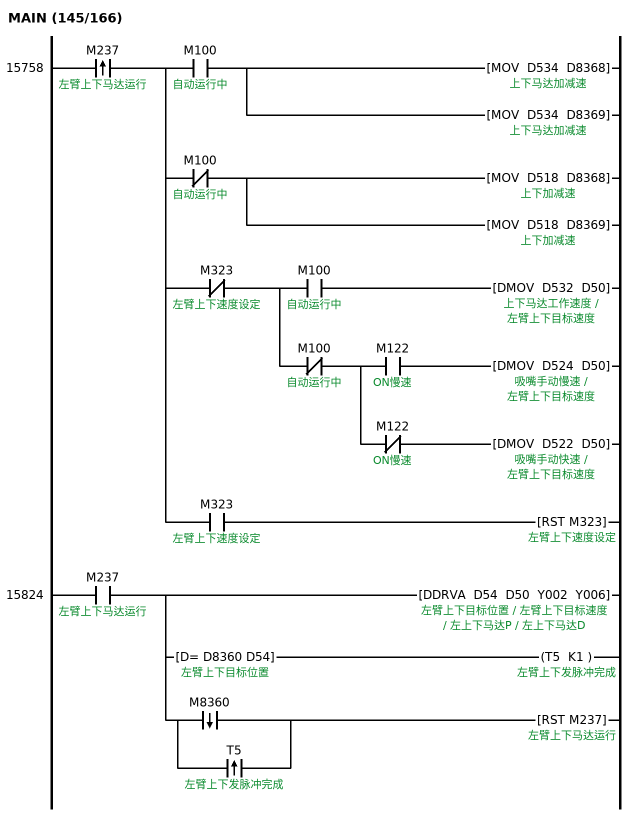
[picture p144: ladder of MAIN, rungs at steps 15758 to 15824]
15758 LDP     M237  ; 左臂上下马达运行
      MPS
      AND     M100  ; 自动运行中
      MOV     D534 D8368
      MOV     D534 D8369
      MRD
      ANI     M100  ; 自动运行中
      MOV     D518 D8368
      MOV     D518 D8369
      MRD
      ANI     M323  ; 左臂上下速度设定
      MPS
      AND     M100  ; 自动运行中
      DMOV    D532 D50
      MPP
      ANI     M100  ; 自动运行中
      MPS
      AND     M122  ; ON慢速
      DMOV    D524 D50
      MPP
      ANI     M122  ; ON慢速
      DMOV    D522 D50
      MPP
      AND     M323  ; 左臂上下速度设定
      RST     M323  ; 左臂上下速度设定
15824 LD      M237  ; 左臂上下马达运行
      DDRVA   D54 D50 Y002 Y006  ; 左上下马达P / 左上下马达D
      MPS
      ANDD=   D8360 D54  ; 左臂上下目标位置
      OUT     T5 K1  ; 左臂上下发脉冲完成
      MPP
      LDF     M8360
      ORP     T5  ; 左臂上下发脉冲完成
      ANB
      RST     M237  ; 左臂上下马达运行
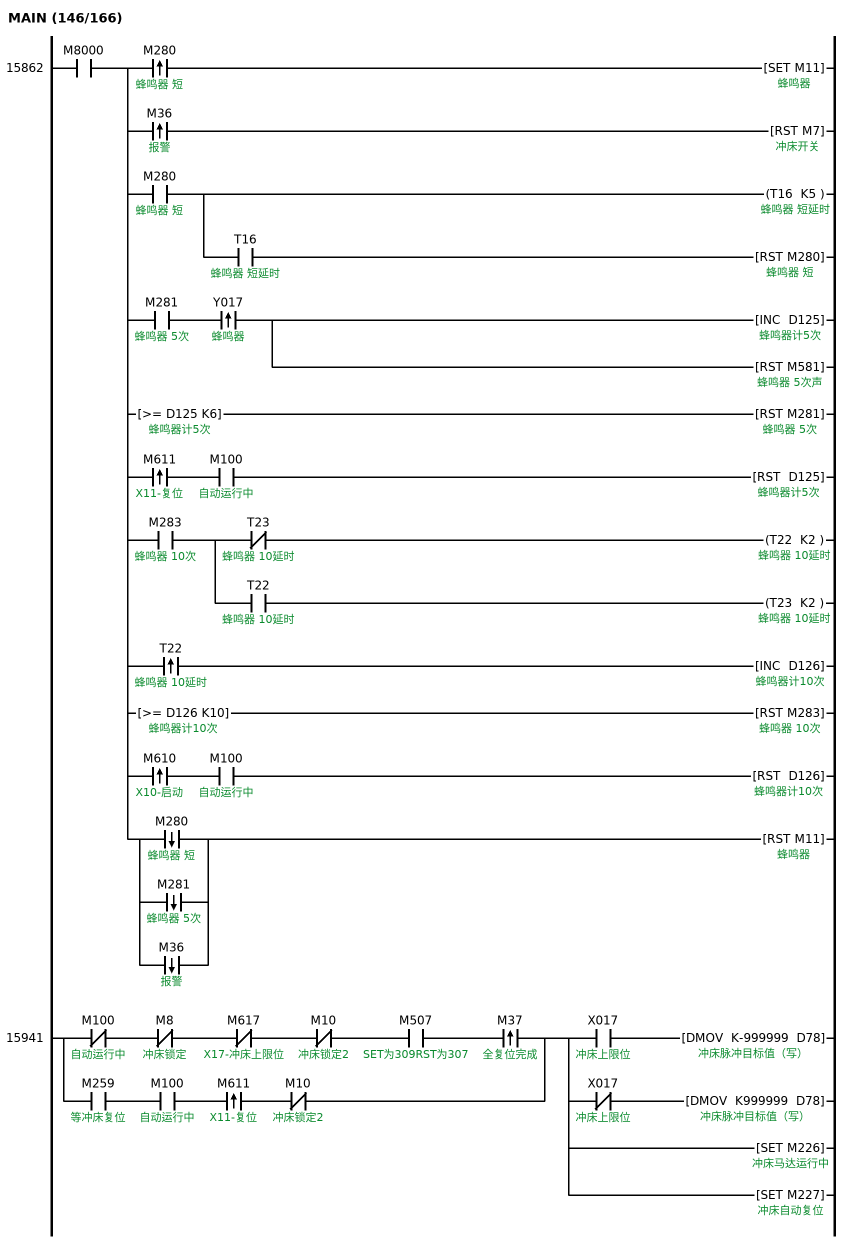
15862 LD      M8000
      MPS
      ANDP    M280  ; 蜂鸣器 短
      SET     M11  ; 蜂鸣器
      MRD
      ANDP    M36  ; 报警
      RST     M7  ; 冲床开关
      MRD
      AND     M280  ; 蜂鸣器 短
      OUT     T16 K5  ; 蜂鸣器 短延时
      AND     T16  ; 蜂鸣器 短延时
      RST     M280  ; 蜂鸣器 短
      MRD
      AND     M281  ; 蜂鸣器 5次
      ANDP    Y017  ; 蜂鸣器
      INC     D125
      RST     M581  ; 蜂鸣器 5次声
      MRD
      AND>=   D125 K6  ; 蜂鸣器计5次
      RST     M281  ; 蜂鸣器 5次
      MRD
      ANDP    M611  ; X11-复位
      AND     M100  ; 自动运行中
      RST     D125  ; 蜂鸣器计5次
      MRD
      AND     M283  ; 蜂鸣器 10次
      MPS
      ANI     T23  ; 蜂鸣器 10延时
      OUT     T22 K2  ; 蜂鸣器 10延时
      MPP
      AND     T22  ; 蜂鸣器 10延时
      OUT     T23 K2  ; 蜂鸣器 10延时
      MRD
      ANDP    T22  ; 蜂鸣器 10延时
      INC     D126  ; 蜂鸣器计10次
      MRD
      AND>=   D126 K10  ; 蜂鸣器计10次
      RST     M283  ; 蜂鸣器 10次
      MRD
      ANDP    M610  ; X10-启动
      AND     M100  ; 自动运行中
      RST     D126  ; 蜂鸣器计10次
      MPP
      LDF     M280  ; 蜂鸣器 短
      ORF     M281  ; 蜂鸣器 5次
      ORF     M36  ; 报警
      ANB
      RST     M11  ; 蜂鸣器
15941 LDI     M100  ; 自动运行中
      ANI     M8  ; 冲床锁定
      ANI     M617  ; X17-冲床上限位
      ANI     M10  ; 冲床锁定2
      AND     M507  ; SET为309RST为307
      ANDP    M37  ; 全复位完成
      LD      M259  ; 等冲床复位
      AND     M100  ; 自动运行中
      ANDP    M611  ; X11-复位
      ANI     M10  ; 冲床锁定2
      ORB
      MPS
      AND     X017  ; 冲床上限位
      DMOV    K-999999 D78  ; 冲床脉冲目标值（写）
      MRD
      ANI     X017  ; 冲床上限位
      DMOV    K999999 D78
      MPP
      SET     M226  ; 冲床马达运行中
      SET     M227  ; 冲床自动复位
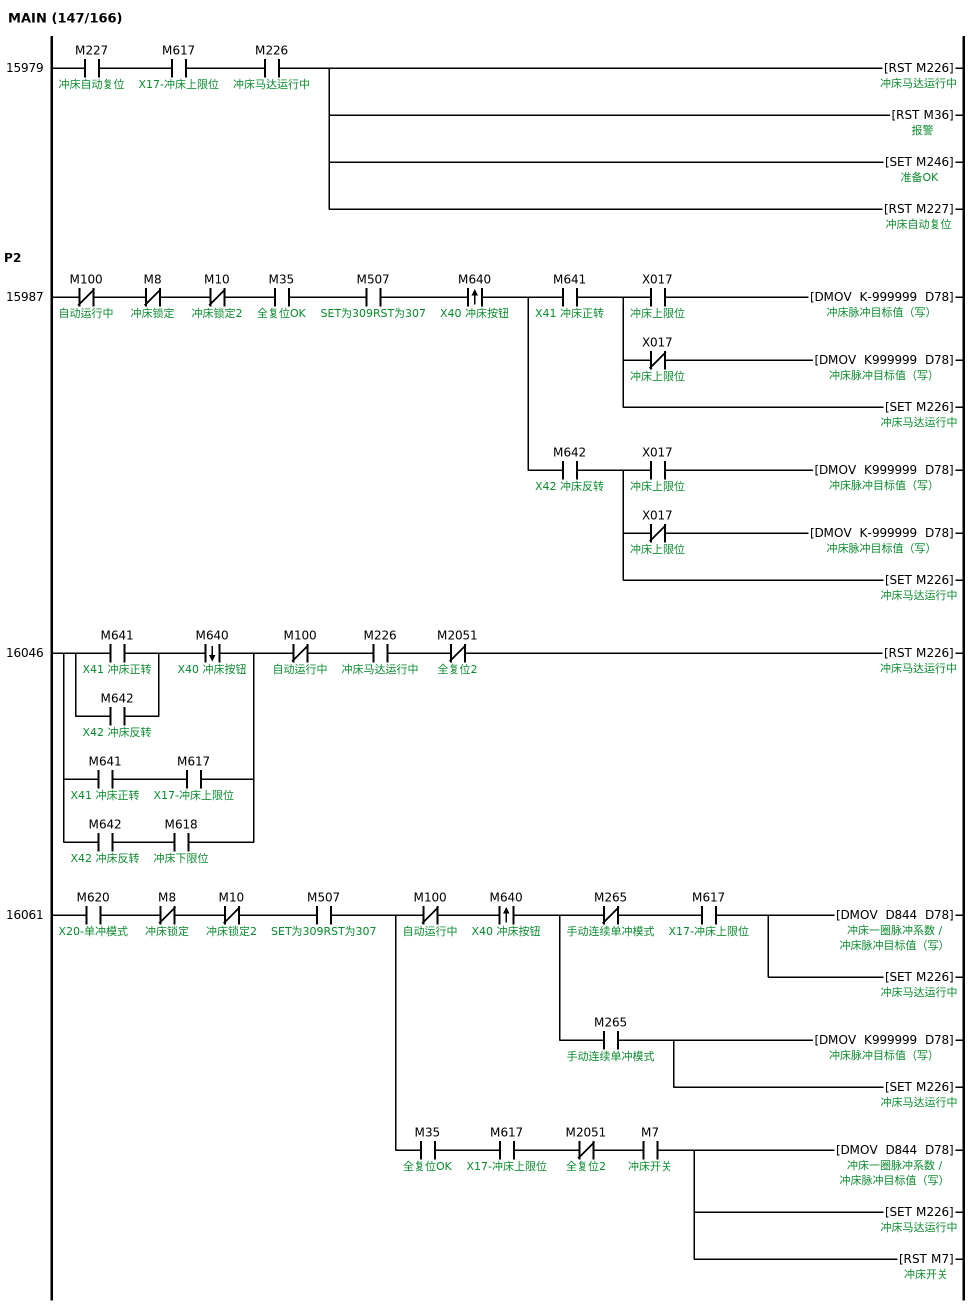
15979 LD      M227  ; 冲床自动复位
      AND     M617  ; X17-冲床上限位
      AND     M226  ; 冲床马达运行中
      RST     M226  ; 冲床马达运行中
      RST     M36  ; 报警
      SET     M246  ; 准备OK
      RST     M227  ; 冲床自动复位
      P2
15987 LDI     M100  ; 自动运行中
      ANI     M8  ; 冲床锁定
      ANI     M10  ; 冲床锁定2
      AND     M35  ; 全复位OK
      AND     M507  ; SET为309RST为307
      ANDP    M640  ; X40 冲床按钮
      MPS
      AND     M641  ; X41 冲床正转
      MPS
      AND     X017  ; 冲床上限位
      DMOV    K-999999 D78
      MRD
      ANI     X017  ; 冲床上限位
      DMOV    K999999 D78
      MPP
      SET     M226  ; 冲床马达运行中
      MPP
      AND     M642  ; X42 冲床反转
      MPS
      AND     X017  ; 冲床上限位
      DMOV    K999999 D78
      MRD
      ANI     X017  ; 冲床上限位
      DMOV    K-999999 D78
      MPP
      SET     M226  ; 冲床马达运行中
16046 LD      M641  ; X41 冲床正转
      OR      M642  ; X42 冲床反转
      ANDF    M640  ; X40 冲床按钮
      LD      M641  ; X41 冲床正转
      AND     M617  ; X17-冲床上限位
      ORB
      LD      M642  ; X42 冲床反转
      AND     M618  ; 冲床下限位
      ORB
      ANI     M100  ; 自动运行中
      AND     M226  ; 冲床马达运行中
      ANI     M2051  ; 全复位2
      RST     M226  ; 冲床马达运行中
16061 LD      M620  ; X20-单冲模式
      ANI     M8  ; 冲床锁定
      ANI     M10  ; 冲床锁定2
      AND     M507  ; SET为309RST为307
      MPS
      ANI     M100  ; 自动运行中
      ANDP    M640  ; X40 冲床按钮
      MPS
      ANI     M265  ; 手动连续单冲模式
      AND     M617  ; X17-冲床上限位
      DMOV    D844 D78
      SET     M226  ; 冲床马达运行中
      MPP
      AND     M265  ; 手动连续单冲模式
      DMOV    K999999 D78
      SET     M226  ; 冲床马达运行中
      MPP
      AND     M35  ; 全复位OK
      AND     M617  ; X17-冲床上限位
      ANI     M2051  ; 全复位2
      AND     M7  ; 冲床开关
      DMOV    D844 D78
      SET     M226  ; 冲床马达运行中
      RST     M7  ; 冲床开关
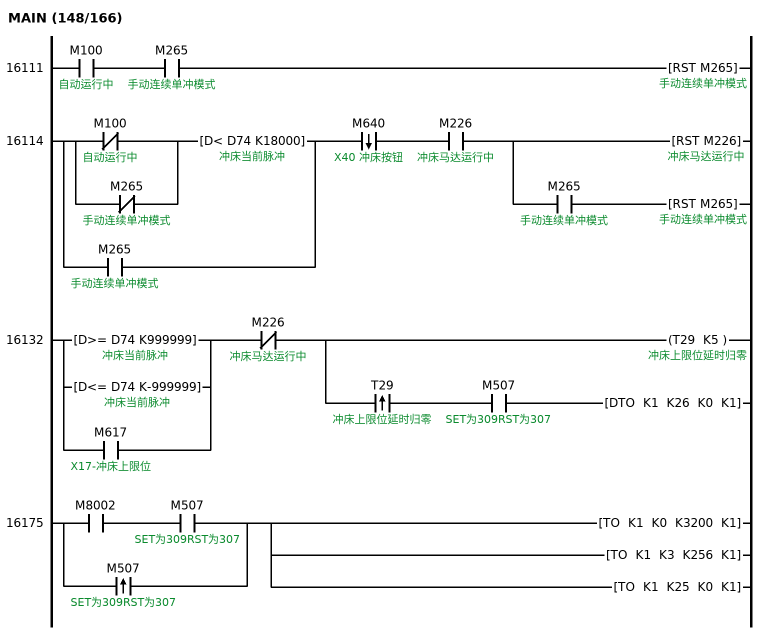
16111 LD      M100  ; 自动运行中
      AND     M265  ; 手动连续单冲模式
      RST     M265  ; 手动连续单冲模式
16114 LDI     M100  ; 自动运行中
      ORI     M265  ; 手动连续单冲模式
      ANDD<   D74 K18000  ; 冲床当前脉冲
      OR      M265  ; 手动连续单冲模式
      ANDF    M640  ; X40 冲床按钮
      AND     M226  ; 冲床马达运行中
      RST     M226  ; 冲床马达运行中
      AND     M265  ; 手动连续单冲模式
      RST     M265  ; 手动连续单冲模式
16132 LDD>=   D74 K999999  ; 冲床当前脉冲
      ORD<=   D74 K-999999  ; 冲床当前脉冲
      OR      M617  ; X17-冲床上限位
      ANI     M226  ; 冲床马达运行中
      OUT     T29 K5  ; 冲床上限位延时归零
      ANDP    T29  ; 冲床上限位延时归零
      AND     M507  ; SET为309RST为307
      DTO     K1 K26 K0 K1
16175 LD      M8002
      AND     M507  ; SET为309RST为307
      ORP     M507  ; SET为309RST为307
      TO      K1 K0 K3200 K1
      TO      K1 K3 K256 K1
      TO      K1 K25 K0 K1
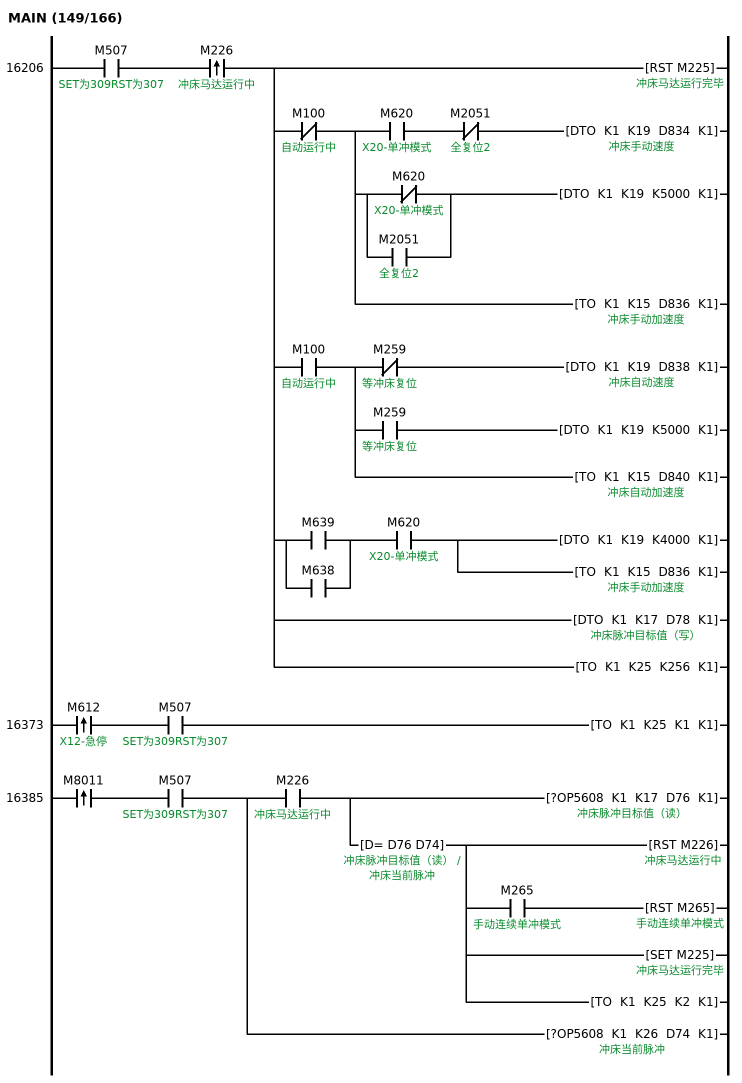
16206 LD      M507  ; SET为309RST为307
      ANDP    M226  ; 冲床马达运行中
      RST     M225  ; 冲床马达运行完毕
      MPS
      ANI     M100  ; 自动运行中
      MPS
      AND     M620  ; X20-单冲模式
      ANI     M2051  ; 全复位2
      DTO     K1 K19 D834 K1
      MRD
      LDI     M620  ; X20-单冲模式
      OR      M2051  ; 全复位2
      ANB
      DTO     K1 K19 K5000 K1
      MPP
      TO      K1 K15 D836 K1
      MRD
      AND     M100  ; 自动运行中
      MPS
      ANI     M259  ; 等冲床复位
      DTO     K1 K19 D838 K1
      MRD
      AND     M259  ; 等冲床复位
      DTO     K1 K19 K5000 K1
      MPP
      TO      K1 K15 D840 K1
      MRD
      LD      M639
      OR      M638
      ANB
      AND     M620  ; X20-单冲模式
      DTO     K1 K19 K4000 K1
      TO      K1 K15 D836 K1
      MPP
      DTO     K1 K17 D78 K1
      TO      K1 K25 K256 K1
16373 LDP     M612  ; X12-急停
      AND     M507  ; SET为309RST为307
      TO      K1 K25 K1 K1
16385 LDP     M8011
      AND     M507  ; SET为309RST为307
      MPS
      AND     M226  ; 冲床马达运行中
      ?OP5608 K1 K17 D76 K1  ; 冲床脉冲目标值（读）
      ANDD=   D76 D74  ; 冲床脉冲目标值（读） / 冲床当前脉冲
      RST     M226  ; 冲床马达运行中
      MPS
      AND     M265  ; 手动连续单冲模式
      RST     M265  ; 手动连续单冲模式
      MPP
      SET     M225  ; 冲床马达运行完毕
      TO      K1 K25 K2 K1
      MPP
      ?OP5608 K1 K26 D74 K1
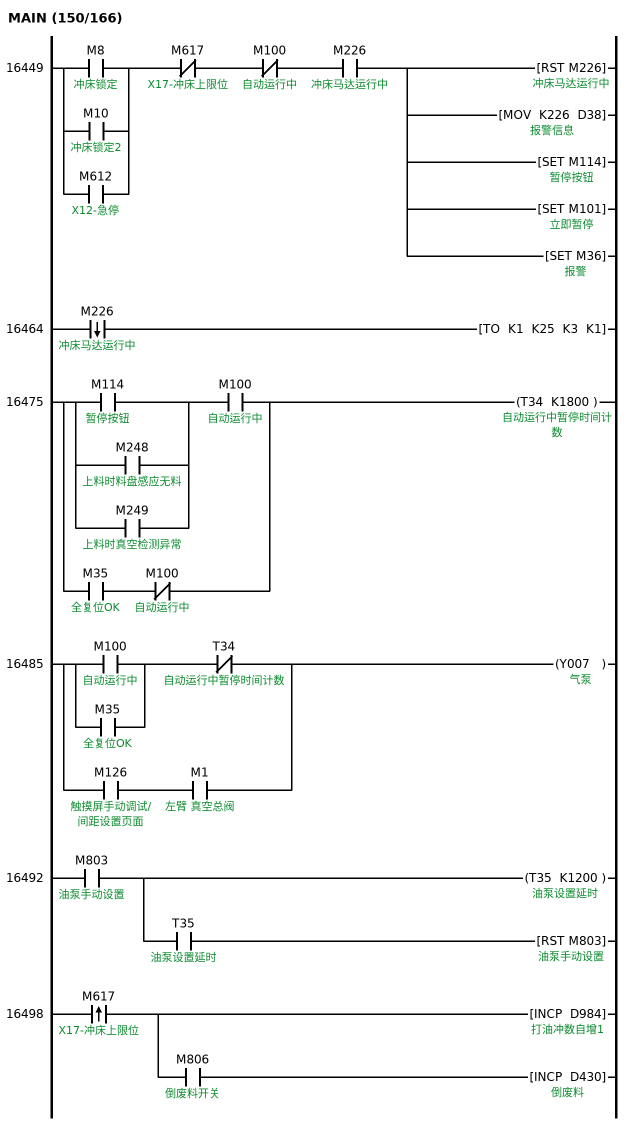
16449 LD      M8  ; 冲床锁定
      OR      M10  ; 冲床锁定2
      OR      M612  ; X12-急停
      ANI     M617  ; X17-冲床上限位
      ANI     M100  ; 自动运行中
      AND     M226  ; 冲床马达运行中
      RST     M226  ; 冲床马达运行中
      MOV     K226 D38
      SET     M114  ; 暂停按钮
      SET     M101  ; 立即暂停
      SET     M36  ; 报警
16464 LDF     M226  ; 冲床马达运行中
      TO      K1 K25 K3 K1
16475 LD      M114  ; 暂停按钮
      OR      M248  ; 上料时料盘感应无料
      OR      M249  ; 上料时真空检测异常
      AND     M100  ; 自动运行中
      LD      M35  ; 全复位OK
      ANI     M100  ; 自动运行中
      ORB
      OUT     T34 K1800  ; 自动运行中暂停时间计数
16485 LD      M100  ; 自动运行中
      OR      M35  ; 全复位OK
      ANI     T34  ; 自动运行中暂停时间计数
      LD      M126  ; 触摸屏手动调试/间距设置页面
      AND     M1  ; 左臂 真空总阀
      ORB
      OUT     Y007  ; 气泵
16492 LD      M803  ; 油泵手动设置
      OUT     T35 K1200  ; 油泵设置延时
      AND     T35  ; 油泵设置延时
      RST     M803  ; 油泵手动设置
16498 LDP     M617  ; X17-冲床上限位
      INCP    D984  ; 打油冲数自增1
      AND     M806  ; 倒废料开关
      INCP    D430  ; 倒废料
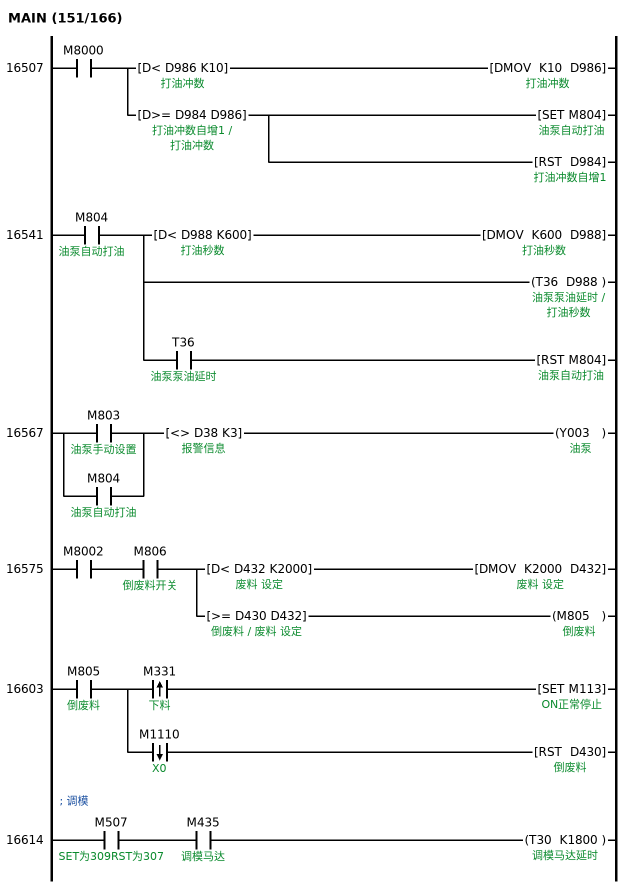
16507 LD      M8000
      MPS
      ANDD<   D986 K10  ; 打油冲数
      DMOV    K10 D986
      MPP
      ANDD>=  D984 D986  ; 打油冲数自增1 / 打油冲数
      SET     M804  ; 油泵自动打油
      RST     D984  ; 打油冲数自增1
16541 LD      M804  ; 油泵自动打油
      MPS
      ANDD<   D988 K600  ; 打油秒数
      DMOV    K600 D988
      MPP
      OUT     T36 D988  ; 油泵泵油延时 / 打油秒数
      AND     T36  ; 油泵泵油延时
      RST     M804  ; 油泵自动打油
16567 LD      M803  ; 油泵手动设置
      OR      M804  ; 油泵自动打油
      AND<>   D38 K3  ; 报警信息
      OUT     Y003  ; 油泵
16575 LD      M8002
      AND     M806  ; 倒废料开关
      MPS
      ANDD<   D432 K2000  ; 废料 设定
      DMOV    K2000 D432
      MPP
      AND>=   D430 D432  ; 倒废料 / 废料 设定
      OUT     M805  ; 倒废料
16603 LD      M805  ; 倒废料
      MPS
      ANDP    M331  ; 下料
      SET     M113  ; ON正常停止
      MPP
      ANDF    M1110  ; X0
      RST     D430  ; 倒废料
; 调模
16614 LD      M507  ; SET为309RST为307
      AND     M435  ; 调模马达
      OUT     T30 K1800  ; 调模马达延时
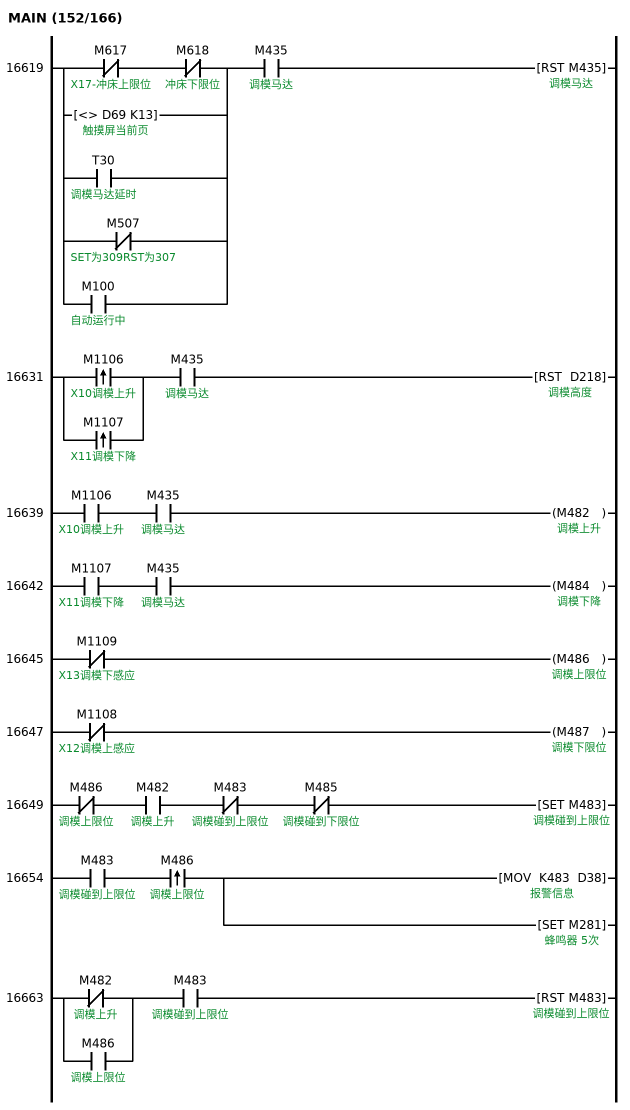
16619 LDI     M617  ; X17-冲床上限位
      ANI     M618  ; 冲床下限位
      OR<>    D69 K13  ; 触摸屏当前页
      OR      T30  ; 调模马达延时
      ORI     M507  ; SET为309RST为307
      OR      M100  ; 自动运行中
      AND     M435  ; 调模马达
      RST     M435  ; 调模马达
16631 LDP     M1106  ; X10调模上升
      ORP     M1107  ; X11调模下降
      AND     M435  ; 调模马达
      RST     D218  ; 调模高度
16639 LD      M1106  ; X10调模上升
      AND     M435  ; 调模马达
      OUT     M482  ; 调模上升
16642 LD      M1107  ; X11调模下降
      AND     M435  ; 调模马达
      OUT     M484  ; 调模下降
16645 LDI     M1109  ; X13调模下感应
      OUT     M486  ; 调模上限位
16647 LDI     M1108  ; X12调模上感应
      OUT     M487  ; 调模下限位
16649 LDI     M486  ; 调模上限位
      AND     M482  ; 调模上升
      ANI     M483  ; 调模碰到上限位
      ANI     M485  ; 调模碰到下限位
      SET     M483  ; 调模碰到上限位
16654 LD      M483  ; 调模碰到上限位
      ANDP    M486  ; 调模上限位
      MOV     K483 D38
      SET     M281  ; 蜂鸣器 5次
16663 LDI     M482  ; 调模上升
      OR      M486  ; 调模上限位
      AND     M483  ; 调模碰到上限位
      RST     M483  ; 调模碰到上限位
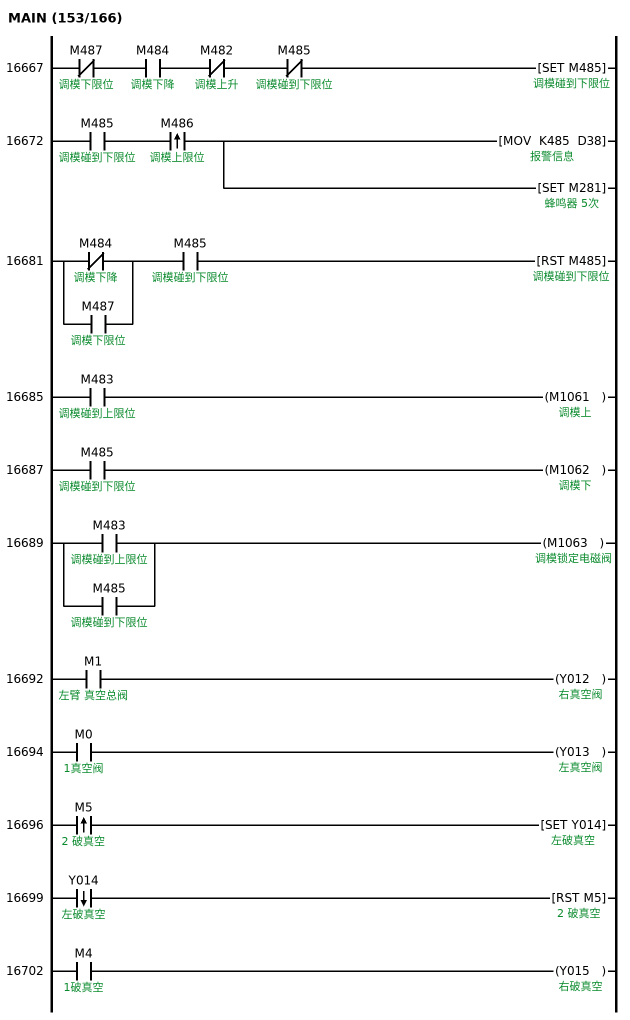
16667 LDI     M487  ; 调模下限位
      AND     M484  ; 调模下降
      ANI     M482  ; 调模上升
      ANI     M485  ; 调模碰到下限位
      SET     M485  ; 调模碰到下限位
16672 LD      M485  ; 调模碰到下限位
      ANDP    M486  ; 调模上限位
      MOV     K485 D38
      SET     M281  ; 蜂鸣器 5次
16681 LDI     M484  ; 调模下降
      OR      M487  ; 调模下限位
      AND     M485  ; 调模碰到下限位
      RST     M485  ; 调模碰到下限位
16685 LD      M483  ; 调模碰到上限位
      OUT     M1061  ; 调模上
16687 LD      M485  ; 调模碰到下限位
      OUT     M1062  ; 调模下
16689 LD      M483  ; 调模碰到上限位
      OR      M485  ; 调模碰到下限位
      OUT     M1063  ; 调模锁定电磁阀
16692 LD      M1  ; 左臂 真空总阀
      OUT     Y012  ; 右真空阀
16694 LD      M0  ; 1真空阀
      OUT     Y013  ; 左真空阀
16696 LDP     M5  ; 2 破真空
      SET     Y014  ; 左破真空
16699 LDF     Y014  ; 左破真空
      RST     M5  ; 2 破真空
16702 LD      M4  ; 1破真空
      OUT     Y015  ; 右破真空
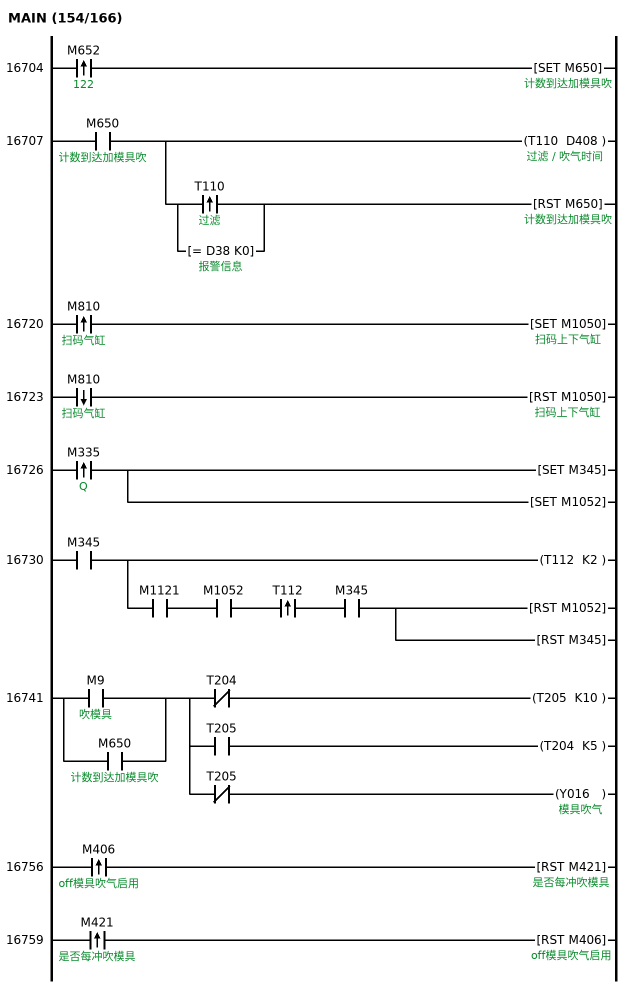
16704 LDP     M652  ; 122
      SET     M650  ; 计数到达加模具吹
16707 LD      M650  ; 计数到达加模具吹
      OUT     T110 D408  ; 过滤 / 吹气时间
      LDP     T110  ; 过滤
      OR=     D38 K0  ; 报警信息
      ANB
      RST     M650  ; 计数到达加模具吹
16720 LDP     M810  ; 扫码气缸
      SET     M1050  ; 扫码上下气缸
16723 LDF     M810  ; 扫码气缸
      RST     M1050  ; 扫码上下气缸
16726 LDP     M335  ; Q
      SET     M345
      SET     M1052
16730 LD      M345
      OUT     T112 K2
      AND     M1121
      AND     M1052
      ANDP    T112
      AND     M345
      RST     M1052
      RST     M345
16741 LD      M9  ; 吹模具
      OR      M650  ; 计数到达加模具吹
      MPS
      ANI     T204
      OUT     T205 K10
      MRD
      AND     T205
      OUT     T204 K5
      MPP
      ANI     T205
      OUT     Y016  ; 模具吹气
16756 LDP     M406  ; off模具吹气启用
      RST     M421  ; 是否每冲吹模具
16759 LDP     M421  ; 是否每冲吹模具
      RST     M406  ; off模具吹气启用
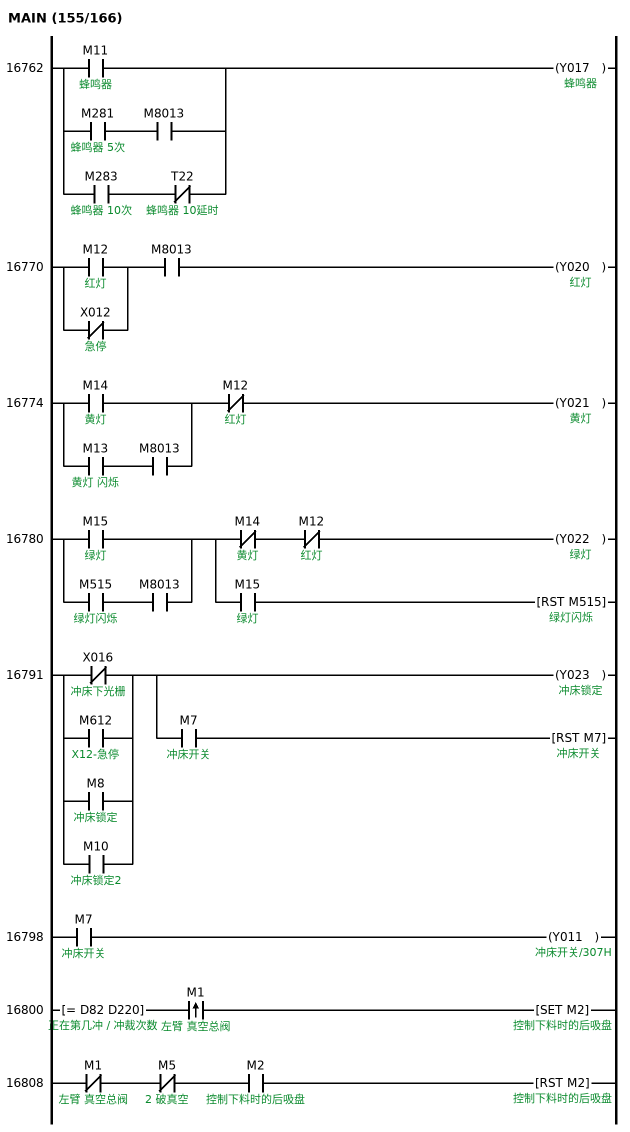
16762 LD      M11  ; 蜂鸣器
      LD      M281  ; 蜂鸣器 5次
      AND     M8013
      ORB
      LD      M283  ; 蜂鸣器 10次
      ANI     T22  ; 蜂鸣器 10延时
      ORB
      OUT     Y017  ; 蜂鸣器
16770 LD      M12  ; 红灯
      ORI     X012  ; 急停
      AND     M8013
      OUT     Y020  ; 红灯
16774 LD      M14  ; 黄灯
      LD      M13  ; 黄灯 闪烁
      AND     M8013
      ORB
      ANI     M12  ; 红灯
      OUT     Y021  ; 黄灯
16780 LD      M15  ; 绿灯
      LD      M515  ; 绿灯闪烁
      AND     M8013
      ORB
      MPS
      ANI     M14  ; 黄灯
      ANI     M12  ; 红灯
      OUT     Y022  ; 绿灯
      MPP
      AND     M15  ; 绿灯
      RST     M515  ; 绿灯闪烁
16791 LDI     X016  ; 冲床下光栅
      OR      M612  ; X12-急停
      OR      M8  ; 冲床锁定
      OR      M10  ; 冲床锁定2
      OUT     Y023  ; 冲床锁定
      AND     M7  ; 冲床开关
      RST     M7  ; 冲床开关
16798 LD      M7  ; 冲床开关
      OUT     Y011  ; 冲床开关/307H
16800 LD=     D82 D220  ; 正在第几冲 / 冲裁次数
      ANDP    M1  ; 左臂 真空总阀
      SET     M2  ; 控制下料时的后吸盘
16808 LDI     M1  ; 左臂 真空总阀
      ANI     M5  ; 2 破真空
      AND     M2  ; 控制下料时的后吸盘
      RST     M2  ; 控制下料时的后吸盘
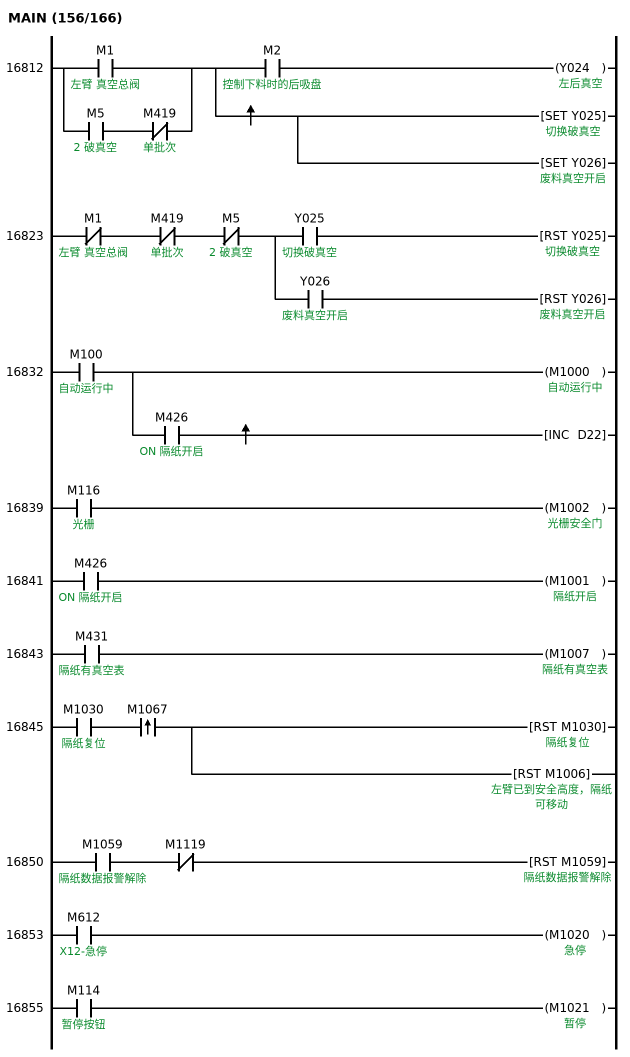
16812 LD      M1  ; 左臂 真空总阀
      LD      M5  ; 2 破真空
      ANI     M419  ; 单批次
      ORB
      MPS
      AND     M2  ; 控制下料时的后吸盘
      OUT     Y024  ; 左后真空
      MPP
      MEP
      SET     Y025  ; 切换破真空
      SET     Y026  ; 废料真空开启
16823 LDI     M1  ; 左臂 真空总阀
      ANI     M419  ; 单批次
      ANI     M5  ; 2 破真空
      MPS
      AND     Y025  ; 切换破真空
      RST     Y025  ; 切换破真空
      MPP
      AND     Y026  ; 废料真空开启
      RST     Y026  ; 废料真空开启
16832 LD      M100  ; 自动运行中
      OUT     M1000  ; 自动运行中
      AND     M426  ; ON 隔纸开启
      MEP
      INC     D22
16839 LD      M116  ; 光栅
      OUT     M1002  ; 光栅安全门
16841 LD      M426  ; ON 隔纸开启
      OUT     M1001  ; 隔纸开启
16843 LD      M431  ; 隔纸有真空表
      OUT     M1007  ; 隔纸有真空表
16845 LD      M1030  ; 隔纸复位
      ANDP    M1067
      RST     M1030  ; 隔纸复位
      RST     M1006  ; 左臂已到安全高度，隔纸可移动
16850 LD      M1059  ; 隔纸数据报警解除
      ANI     M1119
      RST     M1059  ; 隔纸数据报警解除
16853 LD      M612  ; X12-急停
      OUT     M1020  ; 急停
16855 LD      M114  ; 暂停按钮
      OUT     M1021  ; 暂停
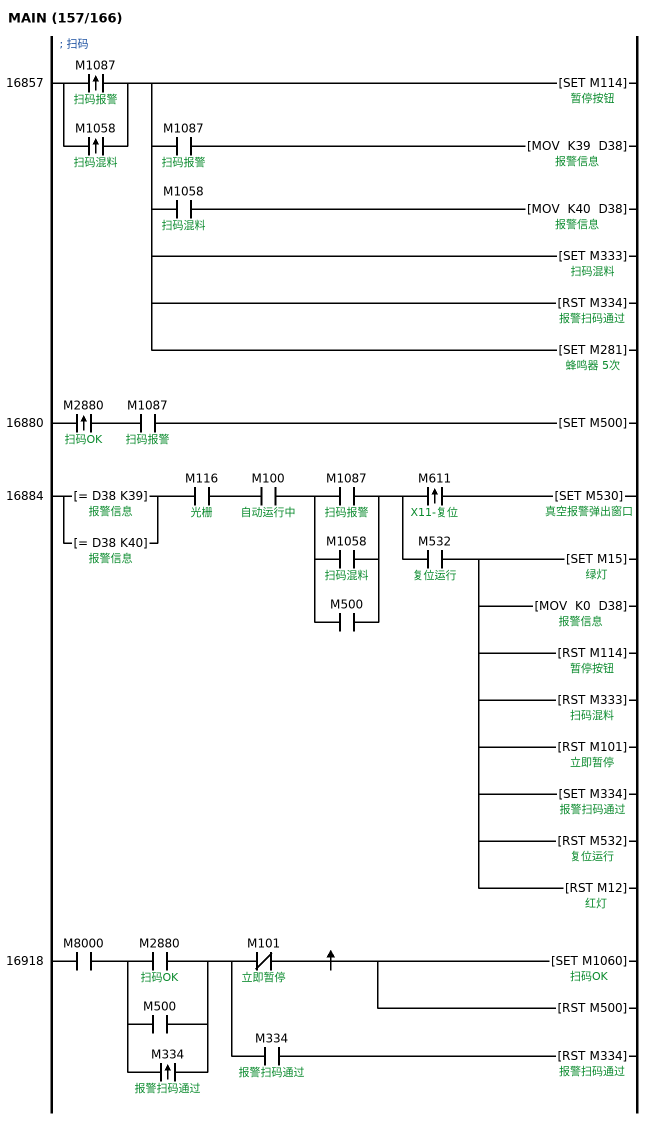
; 扫码
16857 LDP     M1087  ; 扫码报警
      ORP     M1058  ; 扫码混料
      SET     M114  ; 暂停按钮
      MPS
      AND     M1087  ; 扫码报警
      MOV     K39 D38
      MRD
      AND     M1058  ; 扫码混料
      MOV     K40 D38
      MPP
      SET     M333  ; 扫码混料
      RST     M334  ; 报警扫码通过
      SET     M281  ; 蜂鸣器 5次
16880 LDP     M2880  ; 扫码OK
      AND     M1087  ; 扫码报警
      SET     M500
16884 LD=     D38 K39  ; 报警信息
      OR=     D38 K40  ; 报警信息
      AND     M116  ; 光栅
      AND     M100  ; 自动运行中
      LD      M1087  ; 扫码报警
      OR      M1058  ; 扫码混料
      OR      M500
      ANB
      MPS
      ANDP    M611  ; X11-复位
      SET     M530  ; 真空报警弹出窗口
      MPP
      AND     M532  ; 复位运行
      SET     M15  ; 绿灯
      MOV     K0 D38
      RST     M114  ; 暂停按钮
      RST     M333  ; 扫码混料
      RST     M101  ; 立即暂停
      SET     M334  ; 报警扫码通过
      RST     M532  ; 复位运行
      RST     M12  ; 红灯
16918 LD      M8000
      LD      M2880  ; 扫码OK
      OR      M500
      ORP     M334  ; 报警扫码通过
      ANB
      MPS
      ANI     M101  ; 立即暂停
      MEP
      SET     M1060  ; 扫码OK
      RST     M500
      MPP
      AND     M334  ; 报警扫码通过
      RST     M334  ; 报警扫码通过
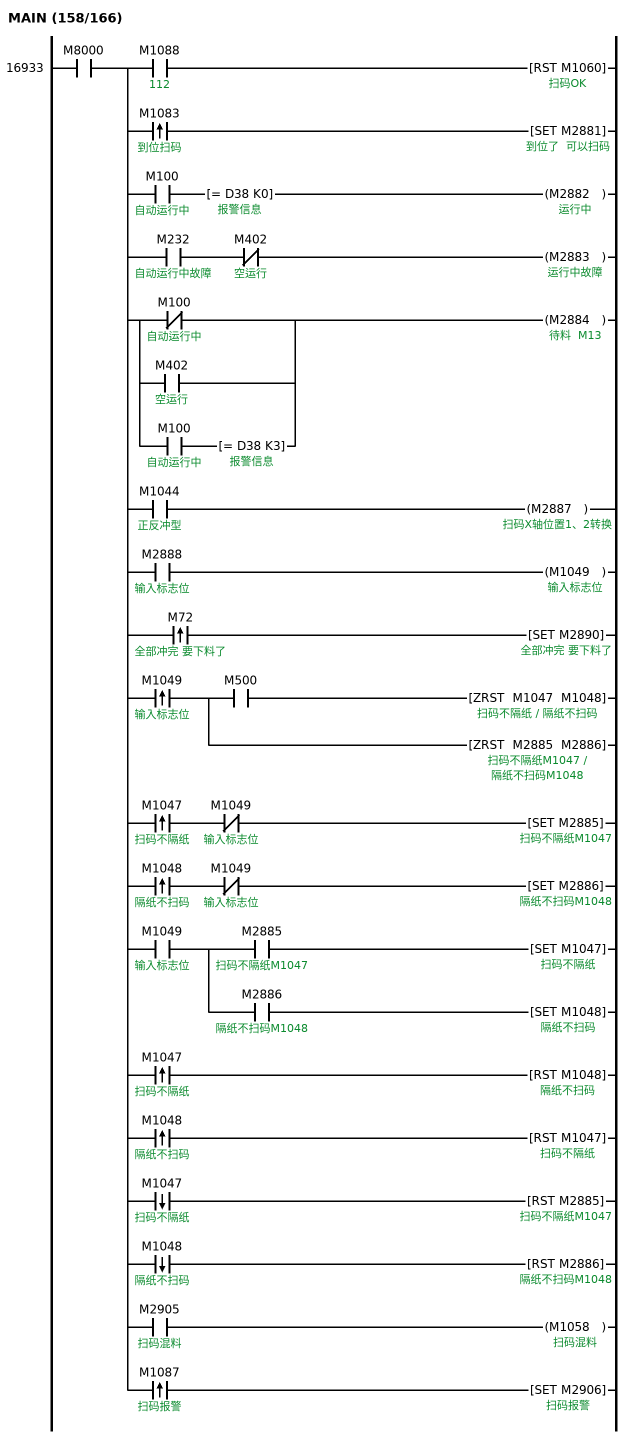
16933 LD      M8000
      MPS
      AND     M1088  ; 112
      RST     M1060  ; 扫码OK
      MRD
      ANDP    M1083  ; 到位扫码
      SET     M2881  ; 到位了  可以扫码
      MRD
      AND     M100  ; 自动运行中
      AND=    D38 K0  ; 报警信息
      OUT     M2882  ; 运行中
      MRD
      AND     M232  ; 自动运行中故障
      ANI     M402  ; 空运行
      OUT     M2883  ; 运行中故障
      MRD
      LDI     M100  ; 自动运行中
      OR      M402  ; 空运行
      LD      M100  ; 自动运行中
      AND=    D38 K3  ; 报警信息
      ORB
      ANB
      OUT     M2884  ; 待料  M13
      MRD
      AND     M1044  ; 正反冲型
      OUT     M2887  ; 扫码X轴位置1、2转换
      MRD
      AND     M2888  ; 输入标志位
      OUT     M1049  ; 输入标志位
      MRD
      ANDP    M72  ; 全部冲完 要下料了
      SET     M2890  ; 全部冲完 要下料了
      MRD
      ANDP    M1049  ; 输入标志位
      MPS
      AND     M500
      ZRST    M1047 M1048
      MPP
      ZRST    M2885 M2886  ; 扫码不隔纸M1047 / 隔纸不扫码M1048
      MRD
      ANDP    M1047  ; 扫码不隔纸
      ANI     M1049  ; 输入标志位
      SET     M2885  ; 扫码不隔纸M1047
      MRD
      ANDP    M1048  ; 隔纸不扫码
      ANI     M1049  ; 输入标志位
      SET     M2886  ; 隔纸不扫码M1048
      MRD
      AND     M1049  ; 输入标志位
      MPS
      AND     M2885  ; 扫码不隔纸M1047
      SET     M1047  ; 扫码不隔纸
      MPP
      AND     M2886  ; 隔纸不扫码M1048
      SET     M1048  ; 隔纸不扫码
      MRD
      ANDP    M1047  ; 扫码不隔纸
      RST     M1048  ; 隔纸不扫码
      MRD
      ANDP    M1048  ; 隔纸不扫码
      RST     M1047  ; 扫码不隔纸
      MRD
      ANDF    M1047  ; 扫码不隔纸
      RST     M2885  ; 扫码不隔纸M1047
      MRD
      ANDF    M1048  ; 隔纸不扫码
      RST     M2886  ; 隔纸不扫码M1048
      MRD
      AND     M2905  ; 扫码混料
      OUT     M1058  ; 扫码混料
      MPP
      ANDP    M1087  ; 扫码报警
      SET     M2906  ; 扫码报警
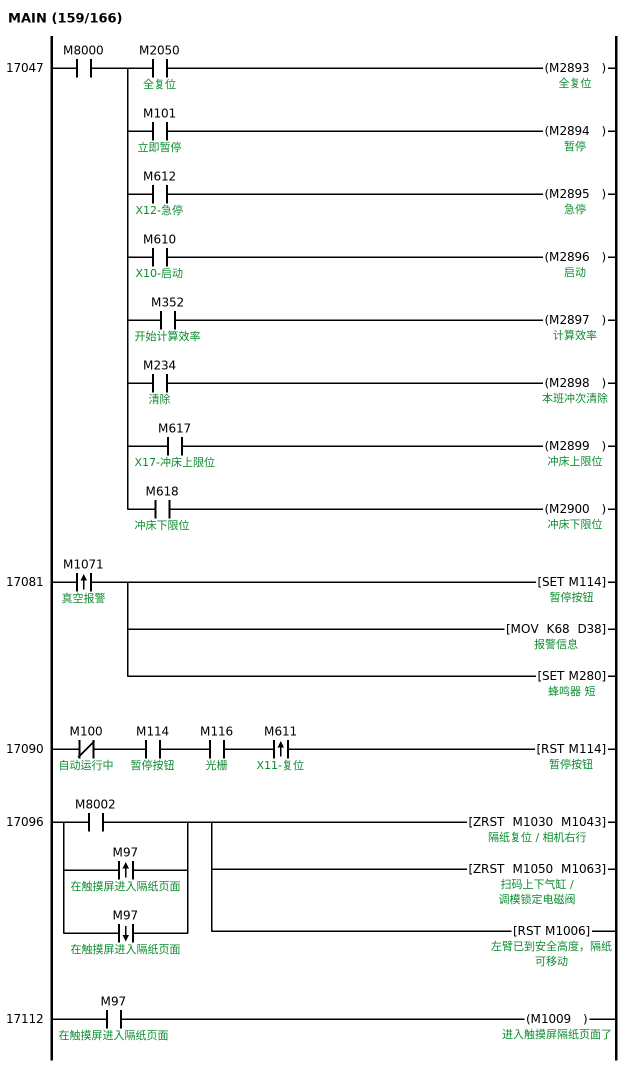
17047 LD      M8000
      MPS
      AND     M2050  ; 全复位
      OUT     M2893  ; 全复位
      MRD
      AND     M101  ; 立即暂停
      OUT     M2894  ; 暂停
      MRD
      AND     M612  ; X12-急停
      OUT     M2895  ; 急停
      MRD
      AND     M610  ; X10-启动
      OUT     M2896  ; 启动
      MRD
      AND     M352  ; 开始计算效率
      OUT     M2897  ; 计算效率
      MRD
      AND     M234  ; 清除
      OUT     M2898  ; 本班冲次清除
      MRD
      AND     M617  ; X17-冲床上限位
      OUT     M2899  ; 冲床上限位
      MPP
      AND     M618  ; 冲床下限位
      OUT     M2900  ; 冲床下限位
17081 LDP     M1071  ; 真空报警
      SET     M114  ; 暂停按钮
      MOV     K68 D38
      SET     M280  ; 蜂鸣器 短
17090 LDI     M100  ; 自动运行中
      AND     M114  ; 暂停按钮
      AND     M116  ; 光栅
      ANDP    M611  ; X11-复位
      RST     M114  ; 暂停按钮
17096 LD      M8002
      ORP     M97  ; 在触摸屏进入隔纸页面
      ORF     M97  ; 在触摸屏进入隔纸页面
      ZRST    M1030 M1043
      ZRST    M1050 M1063
      RST     M1006  ; 左臂已到安全高度，隔纸可移动
17112 LD      M97  ; 在触摸屏进入隔纸页面
      OUT     M1009  ; 进入触摸屏隔纸页面了
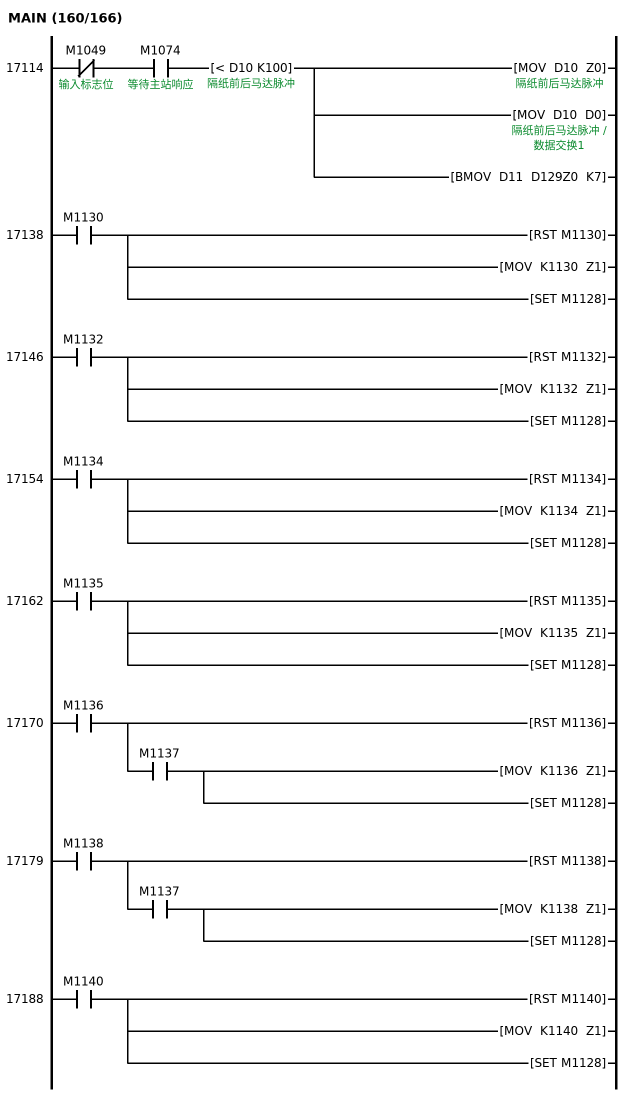
17114 LDI     M1049  ; 输入标志位
      AND     M1074  ; 等待主站响应
      AND<    D10 K100  ; 隔纸前后马达脉冲
      MOV     D10 Z0
      MOV     D10 D0  ; 数据交换1
      BMOV    D11 D129Z0 K7
17138 LD      M1130
      RST     M1130
      MOV     K1130 Z1
      SET     M1128
17146 LD      M1132
      RST     M1132
      MOV     K1132 Z1
      SET     M1128
17154 LD      M1134
      RST     M1134
      MOV     K1134 Z1
      SET     M1128
17162 LD      M1135
      RST     M1135
      MOV     K1135 Z1
      SET     M1128
17170 LD      M1136
      RST     M1136
      AND     M1137
      MOV     K1136 Z1
      SET     M1128
17179 LD      M1138
      RST     M1138
      AND     M1137
      MOV     K1138 Z1
      SET     M1128
17188 LD      M1140
      RST     M1140
      MOV     K1140 Z1
      SET     M1128
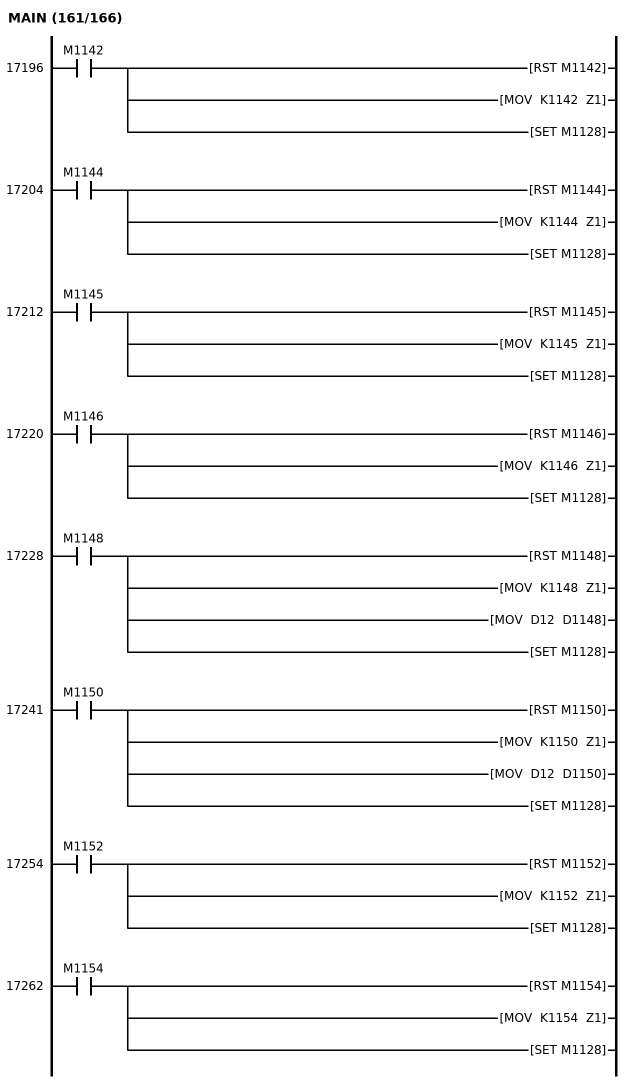
17196 LD      M1142
      RST     M1142
      MOV     K1142 Z1
      SET     M1128
17204 LD      M1144
      RST     M1144
      MOV     K1144 Z1
      SET     M1128
17212 LD      M1145
      RST     M1145
      MOV     K1145 Z1
      SET     M1128
17220 LD      M1146
      RST     M1146
      MOV     K1146 Z1
      SET     M1128
17228 LD      M1148
      RST     M1148
      MOV     K1148 Z1
      MOV     D12 D1148
      SET     M1128
17241 LD      M1150
      RST     M1150
      MOV     K1150 Z1
      MOV     D12 D1150
      SET     M1128
17254 LD      M1152
      RST     M1152
      MOV     K1152 Z1
      SET     M1128
17262 LD      M1154
      RST     M1154
      MOV     K1154 Z1
      SET     M1128
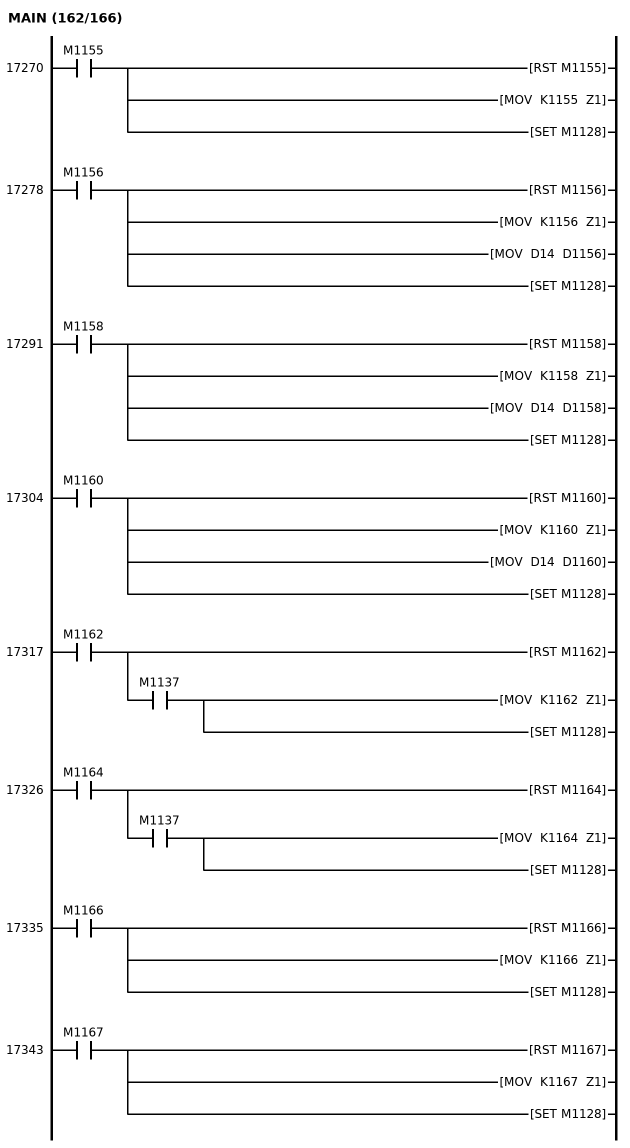
17270 LD      M1155
      RST     M1155
      MOV     K1155 Z1
      SET     M1128
17278 LD      M1156
      RST     M1156
      MOV     K1156 Z1
      MOV     D14 D1156
      SET     M1128
17291 LD      M1158
      RST     M1158
      MOV     K1158 Z1
      MOV     D14 D1158
      SET     M1128
17304 LD      M1160
      RST     M1160
      MOV     K1160 Z1
      MOV     D14 D1160
      SET     M1128
17317 LD      M1162
      RST     M1162
      AND     M1137
      MOV     K1162 Z1
      SET     M1128
17326 LD      M1164
      RST     M1164
      AND     M1137
      MOV     K1164 Z1
      SET     M1128
17335 LD      M1166
      RST     M1166
      MOV     K1166 Z1
      SET     M1128
17343 LD      M1167
      RST     M1167
      MOV     K1167 Z1
      SET     M1128
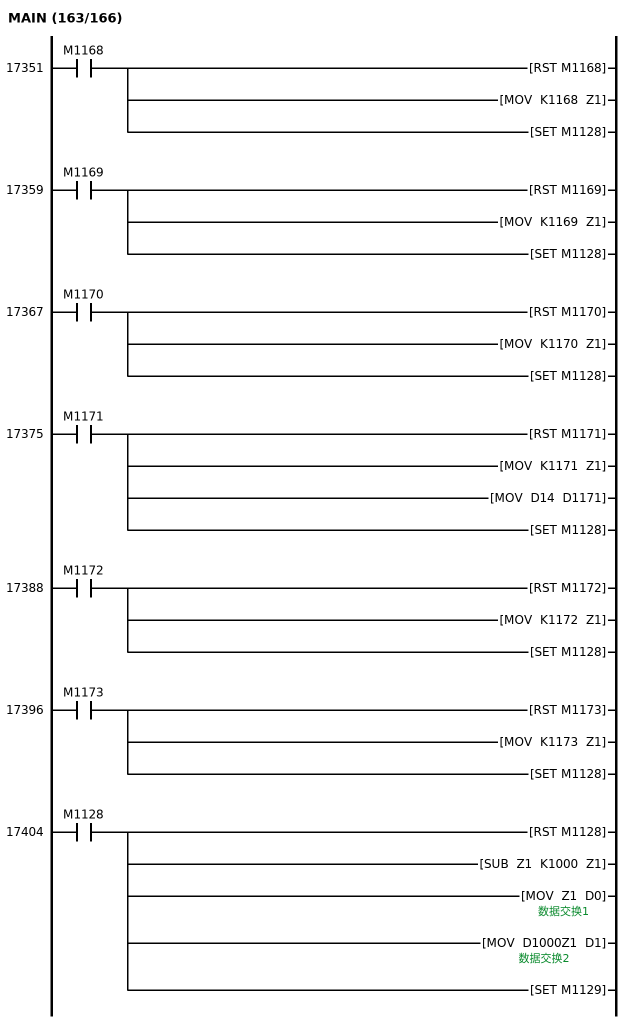
17351 LD      M1168
      RST     M1168
      MOV     K1168 Z1
      SET     M1128
17359 LD      M1169
      RST     M1169
      MOV     K1169 Z1
      SET     M1128
17367 LD      M1170
      RST     M1170
      MOV     K1170 Z1
      SET     M1128
17375 LD      M1171
      RST     M1171
      MOV     K1171 Z1
      MOV     D14 D1171
      SET     M1128
17388 LD      M1172
      RST     M1172
      MOV     K1172 Z1
      SET     M1128
17396 LD      M1173
      RST     M1173
      MOV     K1173 Z1
      SET     M1128
17404 LD      M1128
      RST     M1128
      SUB     Z1 K1000 Z1
      MOV     Z1 D0
      MOV     D1000Z1 D1  ; 数据交换2
      SET     M1129
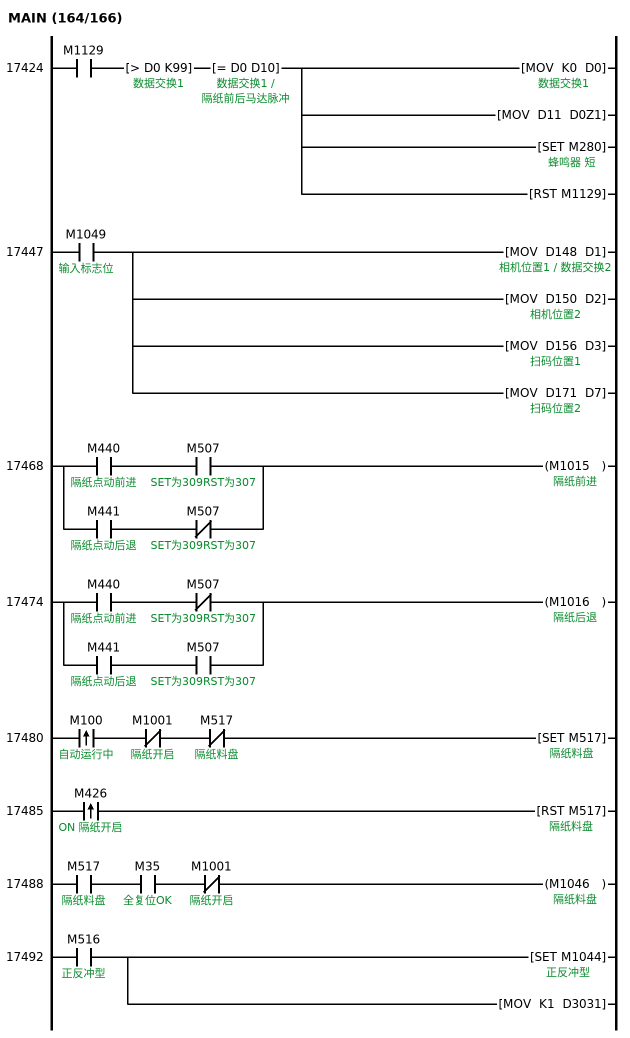
17424 LD      M1129
      AND>    D0 K99  ; 数据交换1
      AND=    D0 D10  ; 数据交换1 / 隔纸前后马达脉冲
      MOV     K0 D0
      MOV     D11 D0Z1
      SET     M280  ; 蜂鸣器 短
      RST     M1129
17447 LD      M1049  ; 输入标志位
      MOV     D148 D1
      MOV     D150 D2
      MOV     D156 D3
      MOV     D171 D7
17468 LD      M440  ; 隔纸点动前进
      AND     M507  ; SET为309RST为307
      LD      M441  ; 隔纸点动后退
      ANI     M507  ; SET为309RST为307
      ORB
      OUT     M1015  ; 隔纸前进
17474 LD      M440  ; 隔纸点动前进
      ANI     M507  ; SET为309RST为307
      LD      M441  ; 隔纸点动后退
      AND     M507  ; SET为309RST为307
      ORB
      OUT     M1016  ; 隔纸后退
17480 LDP     M100  ; 自动运行中
      ANI     M1001  ; 隔纸开启
      ANI     M517  ; 隔纸料盘
      SET     M517  ; 隔纸料盘
17485 LDP     M426  ; ON 隔纸开启
      RST     M517  ; 隔纸料盘
17488 LD      M517  ; 隔纸料盘
      AND     M35  ; 全复位OK
      ANI     M1001  ; 隔纸开启
      OUT     M1046  ; 隔纸料盘
17492 LD      M516  ; 正反冲型
      SET     M1044  ; 正反冲型
      MOV     K1 D3031
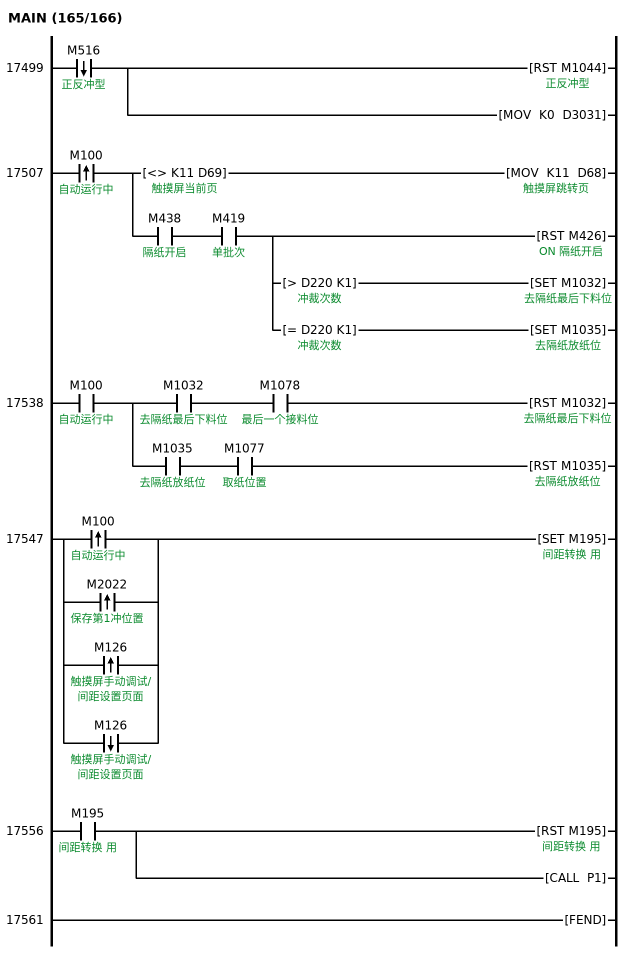
17499 LDF     M516  ; 正反冲型
      RST     M1044  ; 正反冲型
      MOV     K0 D3031
17507 LDP     M100  ; 自动运行中
      MPS
      AND<>   K11 D69  ; 触摸屏当前页
      MOV     K11 D68
      MPP
      AND     M438  ; 隔纸开启
      AND     M419  ; 单批次
      RST     M426  ; ON 隔纸开启
      MPS
      AND>    D220 K1  ; 冲裁次数
      SET     M1032  ; 去隔纸最后下料位
      MPP
      AND=    D220 K1  ; 冲裁次数
      SET     M1035  ; 去隔纸放纸位
17538 LD      M100  ; 自动运行中
      MPS
      AND     M1032  ; 去隔纸最后下料位
      AND     M1078  ; 最后一个接料位
      RST     M1032  ; 去隔纸最后下料位
      MPP
      AND     M1035  ; 去隔纸放纸位
      AND     M1077  ; 取纸位置
      RST     M1035  ; 去隔纸放纸位
17547 LDP     M100  ; 自动运行中
      ORP     M2022  ; 保存第1冲位置
      ORP     M126  ; 触摸屏手动调试/间距设置页面
      ORF     M126  ; 触摸屏手动调试/间距设置页面
      SET     M195  ; 间距转换 用
17556 LD      M195  ; 间距转换 用
      RST     M195  ; 间距转换 用
      CALL    P1
17561 FEND
      P1
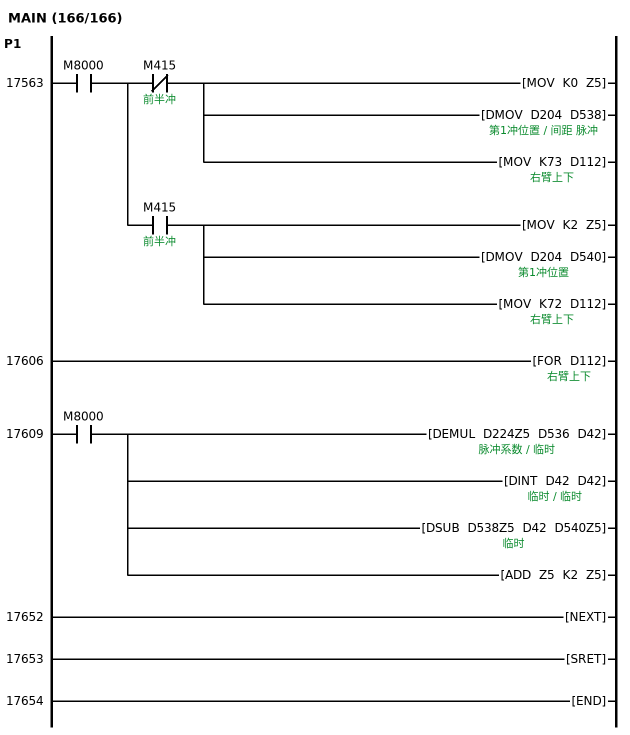
17563 LD      M8000
      MPS
      ANI     M415  ; 前半冲
      MOV     K0 Z5
      DMOV    D204 D538  ; 间距 脉冲
      MOV     K73 D112
      MPP
      AND     M415  ; 前半冲
      MOV     K2 Z5
      DMOV    D204 D540
      MOV     K72 D112
17606 FOR     D112
17609 LD      M8000
      DEMUL   D224Z5 D536 D42
      DINT    D42 D42
      DSUB    D538Z5 D42 D540Z5
      ADD     Z5 K2 Z5
17652 NEXT
17653 SRET
17654 END
END_PROGRAM

// device comments not shown above
M20  ; 可以启动
M29  ; 第1冲已经吸起 是否2冲
M32  ; 下料完成 检查报警信息
M41  ; 前后复位中
M45  ; 清除坐标值
M49  ; 打开文件时处理
M50  ; 取料结束
M51  ; 料盘推高中
M52  ; 二次吸料已开启
M53  ; 推高后回复
M96  ; 没有其他通讯存在
M102  ; 模拟冲床 不开
M112  ; 模拟结束了
M120  ; 右探针 开始检测
M137  ; 等真空后回安全高度
M139  ; 到装模位
M140  ; 等到安全高度
M141  ; 到了安全高度了
M143  ; 到了安全高度
M145  ; 入模 在装模位置了
M146  ; 等破真空
M148  ; 等到安全高度
M149  ; 等到取料位置
M150  ; 再到装模位置
M151  ; 破真空好 上去
M154  ; 再到装模位置
M155  ; 在装模位 到入模
M156  ; 等真空
M157  ; 吸好 上
M163  ; 再到安全位置
M167  ; 到入模高度
M168  ; 等破真空
M169  ; 破真空完 上
M172  ; 等到第一冲位置
M173  ; 到第一冲了 下
M174  ; 等真空
M175  ; 真空吸好 上
M178  ; 再到下料位置
M179  ; 再到下料高度
M189  ; zuo等到安全位置
M190  ; 在下料高度 等破真空
M191  ; 破真空好 上
M192  ; 出模延时 不到第一位置
M196  ; 间距转换 用
M197  ; 真空检测OK
M198  ; 到安全位置
M199  ; 冲完后 上限通了
M202  ; 到装模位置
M203  ; 取料下料
M204  ; 入模
M205  ; 出模
M207  ; 开机不报警
M213  ; 上下限位触发
M216  ; 隔纸机取纸隔料
M217  ; 隔纸机取料移位
M219  ; 下料臂出模 到待模位置中
M220  ; 手动取料时，回安全高度中
M222  ; 上一步状态保存
M223  ; 下料臂 在待模高度
M224  ; 左臂左右正在发脉冲
M228  ; 下料臂待模位置
M229  ; 下料臂到 待模位置
M230  ; 下料臂到安全高度了
M231  ; 下料臂到 待模高度中
M233  ; 到待模高度中
M239  ; 可以到入模位置了
M242  ; 料盘到感应位 OK
M243  ; 料盘到最低位 OK
M244  ; 到 安全高度中
M255  ; 去第一冲中
M260  ; 出模没吸起处理好 启动
M261  ; 报警 2回安全位置
M262  ; 报警 等破真空
M263  ; 第一次启动料盘无料左臂复位
M269  ; 手臂、料盘到位了
M277  ; 取料真空没吸好 1
M278  ; 不抖动 1没吸到 2
M279  ; 抖动2次吸
M284  ; 抖动上 2
M285  ; 抖动 下
M286  ; 抖动完 上了
M287  ; 抖动完 已经上安全高度
M288  ; 抖动 没取到
M289  ; 重复中 抖动时
M314  ; 开机无动作待料状态
M321  ; 料盘速度设定
M324  ; 料盘也要下了
M325  ; 重复 到取料高度开真空
M326  ; 2次到了 开真空
M327  ; 2次 真空开了
M342  ; 单品 退到安全高度了
M346  ; 单品 真空OK
M349  ; ON密码计时
M369  ; zuo延时
M371  ; you磨具针第一次没有检测到
M374  ; 每次吹模具1
M375  ; 等吹气1
M377  ; 每次吹模具2
M378  ; 等吹气2
M397  ; 启动准备
M427  ; 隔纸抖动
M442  ; 保存隔纸长度
M443  ; 保存材料宽度
M444  ; 保存隔料数量
M445  ; 保存抖动频率
M446  ; 保存抖动高度
M447  ; 保存抖动停留时间
M448  ; 保存Y0最大值
M450  ; 保存料盘前后速度
M451  ; 保存料盘手动速度
M452  ; 保存料盘加速度
M521  ; 等装模位置
M522  ; 等入模高度
M523  ; 等探针
M670  ; 扫码上下气缸
M1003  ; 抖动开启
M1004  ; 隔纸复位
M1005  ; 调模上
M1008  ; 隔纸抖动
M1010  ; 到接料位置
M1011  ; 到取纸位置
M1012  ; 到下一料位
M1013  ; 气缸下降
M1014  ; 吸嘴开启
M1017  ; 保存下料中心位
M1018  ; 保存放纸中心位
M1019  ; 取纸隔料
M1022  ; 调模下
M1023  ; 真空检测关闭
M1024  ; 保存Y0最大位置
M1040  ; 相机位置1
M1041  ; 相机位置2
M1042  ; 相机左行
M1045  ; 隔纸前后气缸
M1072  ; 初始化触摸屏数据
M1073  ; 分组传送
M1075  ; 扫码位置2
M1076  ; 前后扫码位置
M1079  ; 倒数第二个接料位
M1080  ; 倒数第三个接料位
M1081  ; 前后最大位置
M1082  ; 前后最小位置
M1084  ; 相机位置1
M1085  ; 相机位置2
M1086  ; 数据输入
M1111  ; X1前后原点
M1112  ; X2上限位
M1113  ; X3
M1114  ; X4真空表
M1115  ; X5下限位
M1124  ; X24右臂探针检测2
M1610  ; 料盘在原点
M1614  ; 计数全复位时模拟复位OK 料盘
M1616  ; 料盘复位清零
M1617  ; 开右中吸嘴
M1618  ; 开右后吸嘴
M2003  ; 下料臂到待模高度
M2004  ; 下料臂 到待模位置
M2007  ; 左臂点动左移
M2008  ; 左臂点动右移
M2017  ; 左臂吸嘴点动下降
M2018  ; 右臂吸嘴点动上升
M2019  ; 上料臂 到待模高度
M2027  ; 保存入模高度
M2046  ; 后真空延时关M16
M2047  ; 上料臂 到待模位置
M2086  ; 料盘最高位设置
M2889  ; 可以启动
M2901  ; 全复位完成
X044  ; 冲床上光栅
X050  ; 上升
X051  ; 下降
X052  ; 调模上限感应器
X053  ; 调模下限感应器
X062  ; 手动料盘上升
X063  ; 手动料盘下降
X064  ; 右臂探针检测2
X066  ; 运行前检测探针
Y030  ; 调模上
Y031  ; 调模下
Y032  ; 调模锁定电磁阀
D15  ; 从站数据交换1
D16  ; 从站数据交换2
D17  ; 从站数据交换3
D28  ; 左臂上下当前值
D36  ; 上下加减速
D80  ; 料盘马达指定速度
D128  ; X100
D130  ; 前后自动速度
D132  ; 前后手动速度
D135  ; 前后停止加速度
D136  ; 前后脉冲系数
D138  ; 上下脉冲系数
D142  ; 上下手动速度
D145  ; 上下停止加速度
D146  ; 上下上升起始慢速
D152  ; 抛纸高度
D154  ; 上升抖动间距
D155  ; 抖动速度
D162  ; 前后最大位置
D164  ; 前后最小位置
D167  ; 隔料间距
D168  ; 气缸抖动频率
D169  ; 气缸抖动时间
D170  ; 慢速上升高度
D172  ; 破真空延时
D173  ; 吸纸真空延时
D412  ; 开机时间累计（分）
D413  ; 开机时间累计（秒）
D414  ; 运行时间累计（分）
D415  ; 运行时间累计（秒）
D416  ; 运行中故障时间（分）
D417  ; 运行中故障时间（秒）
D418  ; 本班冲次
D420  ; 待料时间累计（分）
D421  ; 待料时间累计（秒）
D424  ; 调模高度
D426  ; 机台编号
D428  ; 总冲数
D436  ; 第1料位
D438  ; 第2料位
D440  ; 第3料位
D442  ; 第4料位
D444  ; 第5料位
D446  ; Y0最大位置（写）
D450  ; 上下自动速度（写）
D452  ; 前后自动速度（写）
D454  ; 手动速度（写）
D458  ; 隔纸长度（写）
D460  ; 材料宽度（写）
D462  ; 隔纸数量（写）
D464  ; 抖动频率（写）
D466  ; 抖动高度（写）
D468  ; 停留时间（写）
D470  ; 上下自动速度（读）
D472  ; 前后自动速度（读）
D474  ; 手动速度（读）
D478  ; 隔纸长度（读）
D480  ; 材料宽度（读）
D482  ; 隔纸数量（读）
D484  ; 抖动频率（读）
D486  ; 抖动高度（读）
D488  ; 停留时间（读）
D490  ; 下料中心位（读）
D492  ; 放纸中心位（读）
D494  ; Y0最大位置（读）
D498  ; 当前隔纸位置（mm）
D965  ; 临时2
D967  ; 临时4
T26  ; 红黄灯闪烁
T27  ; 红黄灯闪烁
T37  ; 隔纸延时复位
T52  ; 光栅感应延时1
T53  ; 光栅感应延时2
T80  ; 调模感应断电延时
T107  ; 右臂入模前停留
